PROGRAM MAPPING
VAR
END_VAR

END_PROGRAM

(* stored: Version 1.1.0.1, ProductVersion 3.1.4024.12
   POU MAPPING: Id {e84de69b-ba26-07ad-1592-7be68e226b51}, SpecialFunc None *)
